FUNCTION_BLOCK FB_SLITS_SCATTER EXTENDS FB_SLITS
VAR_INPUT
END_VAR
VAR



END_VAR

END_FUNCTION_BLOCK

(* stored: Version 1.1.0.1, ProductVersion 3.1.4024.6
   POU FB_SLITS_SCATTER: Id {088f7e26-c5bb-497a-8c53-88a89420dd05}, SpecialFunc None *)
